PROGRAM MAIN
VAR
END_VAR

END_PROGRAM

(* stored: Version 1.1.0.1
   POU MAIN: Id {00b5c077-39c9-4b8b-b8f6-f8bd1b09bd42} *)
